(*

short summary
=============

.. <legal notes>

legal notes
=================
| SPDX-FileCopyrightText: © 2023 ekvip automation GmbH <info@ekvip.de>
| SPDX-License-Identifier: Apache-2.0
| For details check: Apache-2.0_

.. _Apache-2.0: https://www.apache.org/licenses/LICENSE-2.0

.. </legal notes>

*)

{warning 'header is generated please add your documentation'}
{attribute 'qualified_only'}
VAR_GLOBAL CONSTANT
	SIZE_OF_ISEQUALTO_DATASET:USINT := 32;
END_VAR

VAR_GLOBAL
	isEqualToDataSetCommon : ARRAY[0..SIZE_OF_ISEQUALTO_DATASET] OF isEqualToDataStr := [
		// test number 0
		( 	StringToTest	:= 'hello',
			WStringToTest	:= "hello",
			EqualToString	:= 'hello',
			EqualToWString	:= "hello",
			IgnoreCases		:= FALSE,
			ExpectedResult	:= FALSE,
			typeToTest		:= TypeToTest.TEST_WSTRING ),

		// test number 1
		( 	StringToTest	:= 'Давным-давно, когда тигр курил',
			WStringToTest	:= "Давным-давно, когда тигр курил",
			EqualToString	:= 'Давным-давно, когда тигр курил',
			EqualToWString	:= "Давным-давно, когда тигр курил",
			IgnoreCases		:= FALSE,
			ExpectedResult	:= FALSE,
			typeToTest		:= TypeToTest.TEST_WSTRING ),
			
		// test number 2
		( 	StringToTest	:= 'לאנג צוריק ווען טיגערס פלעגן רייכערן',
			WStringToTest	:= "לאנג צוריק ווען טיגערס פלעגן רייכערן",
			EqualToString	:= 'לאנג צוריק ווען טיגערס פלעגן רייכערן',
			EqualToWString	:= "לאנג צוריק ווען טיגערס פלעגן רייכערן",
			IgnoreCases		:= FALSE,
			ExpectedResult	:= FALSE,
			typeToTest		:= TypeToTest.TEST_WSTRING ),
			
		// test number 3
		( 	StringToTest	:= 'Давным-давно, когда тигркурил',
			WStringToTest	:= "Давным-давно, когда тигркурил",
			EqualToString	:= 'Давным-давно, когда тигр курил',
			EqualToWString	:= "Давным-давно, когда тигр курил",
			IgnoreCases		:= FALSE,
			ExpectedResult	:= TRUE,
			typeToTest		:= TypeToTest.TEST_WSTRING ),
			
		// test number 4
		( 	StringToTest	:= 'לאנג צוריק ווען טיגערס פלעגןרייכערן',
			WStringToTest	:= "לאנג צוריק ווען טיגערס פלעגןרייכערן",
			EqualToString	:= 'לאנג צוריק ווען טיגערס פלעגן רייכערן',
			EqualToWString	:= "לאנג צוריק ווען טיגערס פלעגן רייכערן",
			IgnoreCases		:= FALSE,
			ExpectedResult	:= TRUE,
			typeToTest		:= TypeToTest.TEST_WSTRING ),
			
		// test number 5
		( 	StringToTest	:= 'לאנג צוריק ווען טיגערס פלעגןרייכערן',
			WStringToTest	:= "לאנג צוריק ווען טיגערס פלעגןרייכערן",
			EqualToString	:= 'לאנג צוריק ווע טיגערס פלעגןרייכערן',
			EqualToWString	:= "לאנג צוריק ווע טיגערס פלעגןרייכערן",
			IgnoreCases		:= FALSE,
			ExpectedResult	:= TRUE,
			typeToTest		:= TypeToTest.TEST_WSTRING ),
			
		// test number 6
		( 	StringToTest	:= '',
			WStringToTest	:= "",
			EqualToString	:= '',
			EqualToWString	:= "",
			IgnoreCases		:= FALSE,
			ExpectedResult	:= FALSE,
			typeToTest		:= TypeToTest.TEST_WSTRING ),
			
		// test number 7
		( 	StringToTest	:= ' ',
			WStringToTest	:= " ",
			EqualToString	:= '  ',
			EqualToWString	:= "  ",
			IgnoreCases		:= FALSE,
			ExpectedResult	:= TRUE,
			typeToTest		:= TypeToTest.TEST_WSTRING ),
			
		// test number 8
		( 	StringToTest	:= 'abc',
			WStringToTest	:= "abc",
			EqualToString	:= 'ABC',
			EqualToWString	:= "ABC",
			IgnoreCases		:= TRUE,
			ExpectedResult	:= FALSE,
			typeToTest		:= TypeToTest.TEST_WSTRING ),

		// test number 9
		( 	StringToTest	:= 'нефти и газа',
			WStringToTest	:= "нефти и газа",
			EqualToString	:= 'НЕФТИ И ГАЗА',
			EqualToWString	:= "НЕФТИ И ГАЗА",
			IgnoreCases		:= TRUE,
			ExpectedResult	:= FALSE,
			typeToTest		:= TypeToTest.TEST_WSTRING ),
		
		// test number 10
		( 	StringToTest	:= 'hello',
			WStringToTest	:= "hello",
			EqualToString	:= 'hello',
			EqualToWString	:= "hello",
			IgnoreCases		:= FALSE,
			ExpectedResult	:= FALSE,
			typeToTest		:= TypeToTest.TEST_STRING ),

		// test number 11
		( 	StringToTest	:= 'Давным-давно, когда тигр курил',
			WStringToTest	:= "Давным-давно, когда тигр курил",
			EqualToString	:= 'Давным-давно, когда тигр курил',
			EqualToWString	:= "Давным-давно, когда тигр курил",
			IgnoreCases		:= FALSE,
			ExpectedResult	:= FALSE,
			typeToTest		:= TypeToTest.TEST_STRING ),
			
		// test number 12
		( 	StringToTest	:= 'לאנג צוריק ווען טיגערס פלעגן רייכערן',
			WStringToTest	:= "לאנג צוריק ווען טיגערס פלעגן רייכערן",
			EqualToString	:= 'לאנג צוריק ווען טיגערס פלעגן רייכערן',
			EqualToWString	:= "לאנג צוריק ווען טיגערס פלעגן רייכערן",
			IgnoreCases		:= FALSE,
			ExpectedResult	:= FALSE,
			typeToTest		:= TypeToTest.TEST_STRING ),
			
		// test number 13
		( 	StringToTest	:= 'Давным-давно, когда тигркурил',
			WStringToTest	:= "Давным-давно, когда тигркурил",
			EqualToString	:= 'Давным-давно, когда тигр курил',
			EqualToWString	:= "Давным-давно, когда тигр курил",
			IgnoreCases		:= FALSE,
			ExpectedResult	:= TRUE,
			typeToTest		:= TypeToTest.TEST_STRING ),
			
		// test number 14
		( 	StringToTest	:= 'לאנג צוריק ווען טיגערס פלעגןרייכערן',
			WStringToTest	:= "לאנג צוריק ווען טיגערס פלעגןרייכערן",
			EqualToString	:= 'לאנג צוריק ווען טיגערס פלעגן רייכערן',
			EqualToWString	:= "לאנג צוריק ווען טיגערס פלעגן רייכערן",
			IgnoreCases		:= FALSE,
			ExpectedResult	:= TRUE,
			typeToTest		:= TypeToTest.TEST_STRING ),
			
		// test number 15
		( 	StringToTest	:= 'לאנג צוריק ווען טיגערס פלעגןרייכערן',
			WStringToTest	:= "לאנג צוריק ווען טיגערס פלעגןרייכערן",
			EqualToString	:= 'לאנג צוריק ווע טיגערס פלעגןרייכערן',
			EqualToWString	:= "לאנג צוריק ווע טיגערס פלעגןרייכערן",
			IgnoreCases		:= FALSE,
			ExpectedResult	:= TRUE,
			typeToTest		:= TypeToTest.TEST_STRING ),
			
		// test number 16
		( 	StringToTest	:= '',
			WStringToTest	:= "",
			EqualToString	:= '',
			EqualToWString	:= "",
			IgnoreCases		:= FALSE,
			ExpectedResult	:= FALSE,
			typeToTest		:= TypeToTest.TEST_STRING ),
			
		// test number 17
		( 	StringToTest	:= ' ',
			WStringToTest	:= " ",
			EqualToString	:= '  ',
			EqualToWString	:= "  ",
			IgnoreCases		:= FALSE,
			ExpectedResult	:= TRUE,
			typeToTest		:= TypeToTest.TEST_STRING ),
			
		// test number 18
		( 	StringToTest	:= 'abc',
			WStringToTest	:= "abc",
			EqualToString	:= 'ABC',
			EqualToWString	:= "ABC",
			IgnoreCases		:= TRUE,
			ExpectedResult	:= FALSE,
			typeToTest		:= TypeToTest.TEST_STRING ),

		// test number 19
		( 	StringToTest	:= 'нефти и газа',
			WStringToTest	:= "нефти и газа",
			EqualToString	:= 'НЕФТИ И ГАЗА',
			EqualToWString	:= "НЕФТИ И ГАЗА",
			IgnoreCases		:= TRUE,
			ExpectedResult	:= FALSE,
			typeToTest		:= TypeToTest.TEST_STRING ),
			
		// test number 20
		( 	StringToTest	:= 'нефти и газа',
			WStringToTest	:= "нефти и газа",
			EqualToString	:= 'НЕФТИ И ГАЗА',
			EqualToWString	:= "НЕФТИ И ГАЗА",
			IgnoreCases		:= TRUE,
			ExpectedResult	:= FALSE,
			typeToTest		:= TypeToTest.TEST_STRING ),

		// test number 21
		( 	StringToTest	:= '',
			WStringToTest	:= "🧐",
			EqualToString	:= '',
			EqualToWString	:= "🧐",
			IgnoreCases		:= TRUE,
			ExpectedResult	:= FALSE,
			typeToTest		:= TypeToTest.TEST_WSTRING ),
			
		// test number 22
		( 	StringToTest	:= '',
			WStringToTest	:= "🧐",
			EqualToString	:= '',
			EqualToWString	:= "🧐",
			IgnoreCases		:= FALSE,
			ExpectedResult	:= FALSE,
			typeToTest		:= TypeToTest.TEST_WSTRING ),
			
		// test number 23
		( 	StringToTest	:= '',
			WStringToTest	:= "h🧐",
			EqualToString	:= '',
			EqualToWString	:= "h🧐",
			IgnoreCases		:= TRUE,
			ExpectedResult	:= FALSE,
			typeToTest		:= TypeToTest.TEST_WSTRING ),
			
		// test number 24
		( 	StringToTest	:= '',
			WStringToTest	:= "h🧐",
			EqualToString	:= '',
			EqualToWString	:= "h🧐",
			IgnoreCases		:= FALSE,
			ExpectedResult	:= FALSE,
			typeToTest		:= TypeToTest.TEST_WSTRING ),
			
		// test number 25
		( 	StringToTest	:= '',
			WStringToTest	:= "h🧐",
			EqualToString	:= '',
			EqualToWString	:= "h🧐 ",
			IgnoreCases		:= TRUE,
			ExpectedResult	:= TRUE,
			typeToTest		:= TypeToTest.TEST_WSTRING ),
			
		// test number 26
		( 	StringToTest	:= '',
			WStringToTest	:= "h🧐",
			EqualToString	:= '',
			EqualToWString	:= "h🧐 ",
			IgnoreCases		:= FALSE,
			ExpectedResult	:= TRUE,
			typeToTest		:= TypeToTest.TEST_WSTRING ),
			
		// test number 27
		( 	StringToTest	:= '$$00434',
			WStringToTest	:= "$$00434",
			EqualToString	:= '$$00434',
			EqualToWString	:= "$$00434",
			IgnoreCases		:= FALSE,
			ExpectedResult	:= FALSE,
			typeToTest		:= TypeToTest.TEST_WSTRING ),
			
		// test number 28
		( 	StringToTest	:= '$$00434',
			WStringToTest	:= "$$00434",
			EqualToString	:= '$$00434',
			EqualToWString	:= "$$00434",
			IgnoreCases		:= TRUE,
			ExpectedResult	:= FALSE,
			typeToTest		:= TypeToTest.TEST_WSTRING ),
			
		// test number 29
		( 	StringToTest	:= '$$00434',
			WStringToTest	:= "$$00434",
			EqualToString	:= '$$00434',
			EqualToWString	:= "$$00434",
			IgnoreCases		:= FALSE,
			ExpectedResult	:= FALSE,
			typeToTest		:= TypeToTest.TEST_STRING ),
			
		// test number 30
		( 	StringToTest	:= '$$00434',
			WStringToTest	:= "$$00434",
			EqualToString	:= '$$00434',
			EqualToWString	:= "$$00434",
			IgnoreCases		:= TRUE,
			ExpectedResult	:= FALSE,
			typeToTest		:= TypeToTest.TEST_STRING ),
			
		// test number 31
		( 	StringToTest	:= '2',
			WStringToTest	:= "2",
			EqualToString	:= '²',
			EqualToWString	:= "²",
			IgnoreCases		:= TRUE,
			ExpectedResult	:= TRUE,
			typeToTest		:= TypeToTest.TEST_STRING ),
			
		// test number 32
		( 	StringToTest	:= '2',
			WStringToTest	:= "2",
			EqualToString	:= '²',
			EqualToWString	:= "²",
			IgnoreCases		:= TRUE,
			ExpectedResult	:= TRUE,
			typeToTest		:= TypeToTest.TEST_WSTRING )
						
	];
END_VAR

(* stored: Version 1.1.0.1, ProductVersion 3.1.4024.12
   GVL isEqualToTestDataSet: Id {e5396f92-a28a-458a-86d3-d12be07b85cf} *)
